// TIA Portal V19 export
TYPE "CTrk_Log"
// stored: Access Published
   STRUCT
      DataValid : Bool;   // Dati registrazione validi
      MES_Received : Bool;   // Dati ricevuti da MES
      MES_Send : Bool;   // Dati inviati a MES
      Logger_Send : Bool;   // Dati inviati a Logger
      O_ID : DInt;   // ID ordine assegnato a bobina
      Diameter : Real;   // Diametro bobina al momento dell'evento
      Tickness : Real;   // Spessore lamiera misurato da sensore al momento dell'evento
      "Tickness_Out-Of-Tol" : Bool;   // Spessore fuori tolleranza
      "DT" : DTL;   // Time stamp al momento dell'evento
   END_STRUCT;
END_TYPE
